FUNCTION_BLOCK DebugInfo
VAR
	_lastMsgIdx			: REFERENCE TO UDINT REF= _Debug.nLastMsg;
	_msg				: REFERENCE TO ARRAY[1..Param.DEBUGMSG_CAP] OF _DebugInfo REF= _Debug.debugMsg;
	
	_lastStrIdx			: REFERENCE TO UDINT REF= _Debug.nLastStr;
	_str				: REFERENCE TO ARRAY[1..Param.DEBUGSTR_CAP] OF Str REF= _Debug.debugStr;
END_VAR

END_FUNCTION_BLOCK

(* stored: Version 1.1.0.1
   POU DebugInfo: Id {489c56af-ae27-4926-af44-96228e2f35be}, SpecialFunc None *)
